(* CoDeSys 2.3.9.55 project: paternoster.pro *)
(* Libraries: Standard.lib*2.6.14 10:37:46, IecSfc.lib*2.6.14 10:37:46 *)

(* Global variable list: Global_Variables *)
VAR_GLOBAL
   (*Entradas *)
      (* Sensores de posición en plantas *)
      S0_1: BOOL;
      S1_1: BOOL;
      S2_1: BOOL;
      S3_1: BOOL;
      S0_2: BOOL;
      S1_2: BOOL;
      S2_2: BOOL;
      S3_2: BOOL;
      (* Pulsadores de llamadas en planta *)
      P0: BOOL;
      P1: BOOL;
      P2: BOOL;
      P3: BOOL;
    (* Pulsadores en cabina  *)
      C0_1: BOOL;
      C1_1: BOOL;
      C2_1: BOOL;
      C3_1: BOOL;
      C0_2: BOOL;
      C1_2: BOOL;
      C2_2: BOOL;
      C3_2: BOOL;
   (*Salidas *)
      Motor_arriba_1 : BOOL;
      Motor_Abajo_1 : BOOL;
     Motor_arriba_2 : BOOL;
      Motor_Abajo_2 : BOOL;
   (* luces asociadas a los pulsadores. Se usarán
        si se quiere implementar memoria de llamada *)
     LuzP0:BOOL;
     LuzP1:BOOL;
     LuzP2:BOOL;
     LuzP3:BOOL;
     LuzC0_1:BOOL;
     LuzC1_1:BOOL;
     LuzC2_1:BOOL;
     LuzC3_1:BOOL;
     LuzC0_2:BOOL;
     LuzC1_2:BOOL;
     LuzC2_2:BOOL;
     LuzC3_2:BOOL;
END_VAR

(* POU PLC_PRG, ST *)
PROGRAM PLC_PRG
VAR
END_VAR
Movimiento1;
Movimiento2;
END_PROGRAM

(* POU Movimiento1, ST *)
PROGRAM Movimiento1
VAR
    pos1:INT:=0;
END_VAR
IF (Motor_arriba_1 AND pos1>=-240) THEN
   pos1:=pos1-2;
END_IF


IF (Motor_abajo_1 AND pos1<=-2) THEN
   pos1:=pos1+2;
END_IF

IF (pos1>=0 AND pos1<=2) THEN
  S0_1:=TRUE;
ELSE
  S0_1:=FALSE;
END_IF

IF (pos1>=-78 AND pos1<=-74) THEN
  S1_1:=TRUE;
ELSE
  S1_1:=FALSE;
END_IF

IF (pos1>=-156 AND pos1<=-152) THEN
  S2_1:=TRUE;
ELSE
  S2_1:=FALSE;
END_IF

IF (pos1>=-242 AND pos1<=-240) THEN
  S3_1:=TRUE;
ELSE
  S3_1:=FALSE;
END_IF
END_PROGRAM

(* POU Movimiento2, ST *)
PROGRAM Movimiento2
VAR
    pos2:INT:=0;
END_VAR
IF (Motor_arriba_2 AND pos2>=-240) THEN
   pos2:=pos2-2;
END_IF


IF (Motor_abajo_2 AND pos2<=-2) THEN
   pos2:=pos2+2;
END_IF

IF (pos2>=0 AND pos2<=2) THEN
  S0_2:=TRUE;
ELSE
  S0_2:=FALSE;
END_IF

IF (pos2>=-78 AND pos2<=-74) THEN
  S1_2:=TRUE;
ELSE
  S1_2:=FALSE;
END_IF

IF (pos2>=-156 AND pos2<=-152) THEN
  S2_2:=TRUE;
ELSE
  S2_2:=FALSE;
END_IF

IF (pos2>=-242 AND pos2<=-240) THEN
  S3_2:=TRUE;
ELSE
  S3_2:=FALSE;
END_IF
END_PROGRAM

(* Visualisation Ascensor
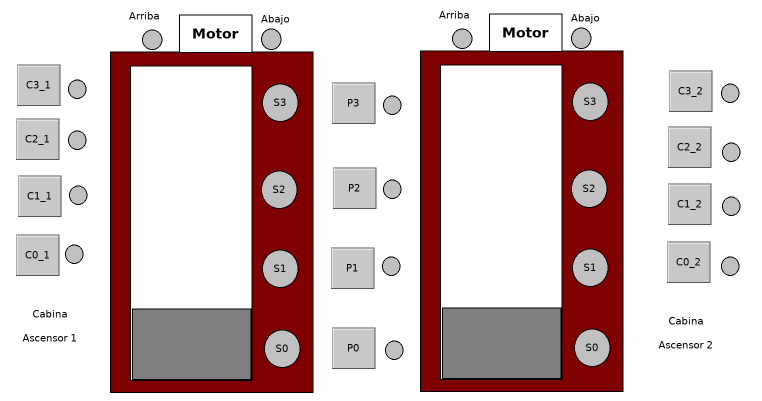
ellipse at (285,341)-(321,379): text "S0"; alarm colour if S0_1
ellipse at (283,261)-(319,299): text "S1"; alarm colour if S1_1
ellipse at (282,182)-(318,220): text "S2"; alarm colour if S2_1
ellipse at (283,95)-(319,133): text "S3"; alarm colour if S3_1
rounded rectangle at (153,320)-(272,391): y offset Movimiento1.pos1
button at (353,339)-(396,380): text "P0"; taps P0
button at (352,259)-(395,300): text "P1"; taps P1
button at (354,179)-(397,220): text "P2"; taps P2
button at (353,94)-(396,135): text "P3"; taps P3
rectangle at (200,26)-(273,64): text "Motor"
ellipse at (163,41)-(183,61): alarm colour if Motor_arriba_1
ellipse at (282,40)-(302,61): alarm colour if Motor_abajo_1
rectangle at (138,18)-(193,37): text "Arriba"
rectangle at (269,21)-(324,40): text "Abajo"
ellipse at (595,340)-(631,378): text "S0"; alarm colour if S0_2
ellipse at (593,260)-(629,298): text "S1"; alarm colour if S1_2
ellipse at (592,181)-(628,219): text "S2"; alarm colour if S2_2
ellipse at (593,94)-(629,132): text "S3"; alarm colour if S3_2
rounded rectangle at (463,319)-(582,390): y offset Movimiento2.pos2
rectangle at (510,25)-(583,63): text "Motor"
ellipse at (473,40)-(493,60): alarm colour if Motor_arriba_2
ellipse at (592,39)-(612,60): alarm colour if Motor_abajo_2
rectangle at (448,17)-(503,36): text "Arriba"
rectangle at (579,20)-(634,39): text "Abajo"
button at (37,246)-(80,287): text "C0_1"; taps C0_1
button at (39,187)-(82,228): text "C1_1"; taps C1_1
button at (37,130)-(80,171): text "C2_1"; taps C2_1
button at (38,76)-(81,117): text "C3_1"; taps C3_1
rectangle at (28,305)-(114,346): text "Cabina"
rectangle at (28,329)-(114,370): text "Ascensor 1"
button at (688,253)-(731,294): text "C0_2"; taps C0_2
button at (689,195)-(732,236): text "C1_2"; taps C1_2
button at (689,138)-(732,179): text "C2_2"; taps C2_2
button at (690,82)-(733,123): text "C3_2"; taps C3_2
rectangle at (664,312)-(750,353): text "Cabina"
rectangle at (664,336)-(750,377): text "Ascensor 2"
ellipse at (89,91)-(107,110): alarm colour if LuzC3_1
ellipse at (89,142)-(107,161): alarm colour if LuzC2_1
ellipse at (90,197)-(108,216): alarm colour if LuzC1_1
ellipse at (86,256)-(104,275): alarm colour if LuzC0_1
ellipse at (404,107)-(422,126): alarm colour if LuzP3
ellipse at (404,191)-(422,210): alarm colour if LuzP2
ellipse at (403,268)-(421,287): alarm colour if LuzP1
ellipse at (406,352)-(424,371): alarm colour if LuzP0
ellipse at (742,95)-(760,114): alarm colour if LuzC3_2
ellipse at (743,154)-(761,173): alarm colour if LuzC2_2
ellipse at (743,208)-(761,227): alarm colour if LuzC1_2
ellipse at (742,268)-(760,287): alarm colour if LuzC0_2
6 more shapes without text or variables
*)
